// TIA Portal V16 export
// export: Created 2024-09-05T17:39:12.5403841Z, ExportSetting WithDefaults, DisplayName Totally Integrated Automation Portal, DisplayVersion V16 Update 6, DisplayName TIA Portal Version Control Interface, DisplayVersion V16 Update 2, DisplayName TIA Portal Openness, DisplayVersion V16 Update 6, DisplayName STEP 7 Professional, DisplayVersion V16 Update 6, DisplayName STEP 7 Safety, DisplayVersion V16, DisplayName WinCC Advanced, DisplayVersion V16 Update 6
DATA_BLOCK "RivetingHistoryLeft_DB"   // DB41
VERSION : 0.1
// stored: AutoNumber true, DBAccessibleFromOPCUA true, InstanceOfName RivetingHistory, InstanceOfType FB
"RivetingHistory"
   // VAR_INPUT
   //    iNewCycle : Bool;
   //    iData : "UDT_Friedrich";
   // END_VAR
   // VAR RETAIN
   //    history : Array[0..99] of "UDT_Friedrich";
   // END_VAR
   // VAR
   //    pageData { S7_SetPoint := 'True'} : Array[0..9] of "UDT_Friedrich";
   // END_VAR
   // VAR RETAIN
   //    pageNumber { S7_SetPoint := 'True'} : USInt := 0;
   // END_VAR
   // VAR
   //    resetHistory : Bool;
   // END_VAR
BEGIN
   history[0..99].Start := FALSE;
   history[0..24].PrgNumber := 2;
   history[25..99].PrgNumber := 0;
   history[0..14].Ready := TRUE;
   history[15].Ready := FALSE;
   history[16..24].Ready := TRUE;
   history[25..99].Ready := FALSE;
   history[0..99].Running := FALSE;
   history[0..4].OK := TRUE;
   history[5..9].OK := FALSE;
   history[10..11].OK := TRUE;
   history[12..13].OK := FALSE;
   history[14..24].OK := TRUE;
   history[25..99].OK := FALSE;
   history[0..4].NOK := FALSE;
   history[5..9].NOK := TRUE;
   history[10..11].NOK := FALSE;
   history[12..13].NOK := TRUE;
   history[14..99].NOK := FALSE;
   history[0..24].H1OK := TRUE;
   history[25..99].H1OK := FALSE;
   history[0..4].H2OK := TRUE;
   history[5..9].H2OK := FALSE;
   history[10..11].H2OK := TRUE;
   history[12..13].H2OK := FALSE;
   history[14..24].H2OK := TRUE;
   history[25..99].H2OK := FALSE;
   history[0..4].TimeOK := TRUE;
   history[5..9].TimeOK := FALSE;
   history[10..11].TimeOK := TRUE;
   history[12..13].TimeOK := FALSE;
   history[14..24].TimeOK := TRUE;
   history[25..99].TimeOK := FALSE;
   history[0..99].StartError := FALSE;
   history[0..99].LastH1 := 0.0;
   history[0..3].LastH2 := 0.0;
   history[4].LastH2 := 2.23;
   history[5..9].LastH2 := 0.0;
   history[10].LastH2 := 2.29;
   history[11].LastH2 := 2.22;
   history[12..13].LastH2 := 0.0;
   history[14].LastH2 := 2.27;
   history[15..16].LastH2 := 2.25;
   history[17].LastH2 := 2.4;
   history[18].LastH2 := 2.28;
   history[19].LastH2 := 2.39;
   history[20].LastH2 := 2.4;
   history[21].LastH2 := 2.39;
   history[22].LastH2 := 2.37;
   history[23..24].LastH2 := 2.4;
   history[25..99].LastH2 := 0.0;
   history[0..18].LastTime := 0.0;
   history[19..21].LastTime := 0.12;
   history[22..23].LastTime := 0.0;
   history[24].LastTime := 0.12;
   history[25..99].LastTime := 0.0;
   history[0].LastZ1 := 11.69;
   history[1].LastZ1 := 11.86;
   history[2].LastZ1 := 11.77;
   history[3].LastZ1 := 11.85;
   history[4].LastZ1 := 12.06;
   history[5].LastZ1 := 11.86;
   history[6].LastZ1 := 11.68;
   history[7].LastZ1 := 11.85;
   history[8].LastZ1 := 11.74;
   history[9].LastZ1 := 11.89;
   history[10].LastZ1 := 12.16;
   history[11].LastZ1 := 12.09;
   history[12].LastZ1 := 11.76;
   history[13].LastZ1 := 11.73;
   history[14].LastZ1 := 12.09;
   history[15..16].LastZ1 := 12.38;
   history[17].LastZ1 := 12.19;
   history[18].LastZ1 := 12.4;
   history[19..24].LastZ1 := 12.2;
   history[25..99].LastZ1 := 0.0;
   history[0..99].Error := FALSE;
   history[0..99].NewData := FALSE;
   history[0..4].Z1OK := TRUE;
   history[5..9].Z1OK := FALSE;
   history[10..11].Z1OK := TRUE;
   history[12..13].Z1OK := FALSE;
   history[14..24].Z1OK := TRUE;
   history[25..99].Z1OK := FALSE;
   history[0..24].NewDataAfterStart := TRUE;
   history[25..99].NewDataAfterStart := FALSE;
   history[0].LastZ2 := 11.69;
   history[1].LastZ2 := 11.86;
   history[2].LastZ2 := 11.77;
   history[3].LastZ2 := 11.85;
   history[4..99].LastZ2 := 0.0;
END_DATA_BLOCK
